// TwinCAT 3 PLC project Main
// ProgramVersion: 3.1.4023.0
// libraries:
//   mobject-fsm, * (mobject-io-ext)
//   Tc3_Module, * (Beckhoff Automation GmbH)
// project tree:
//   / PlcTask.TcTTO
//   Programs/ Main.TcPOU
//   TestMachine/ TestMachine.TcPOU, TestMachineEvents.TcDUT
// real-time tasks:
//   TASK PlcTask: cycle T#10ms, priority 20, ADS port 350

CONFIGURATION Main
    RESOURCE PLC ON TwinCAT3
        TASK PlcTask(INTERVAL := T#10ms, PRIORITY := 20);
        PROGRAM Main WITH PlcTask : Main;
    END_RESOURCE
END_CONFIGURATION

// ---- TestMachine/TestMachineEvents.TcDUT
{attribute 'qualified_only'}
{attribute 'strict'}
TYPE TestMachineEvents :
(
	Start,
	Stop,
	Abort,
	Reset,
	Clear
);
END_TYPE

// ---- Programs/Main.TcPOU
PROGRAM Main
VAR
	machine : TestMachine;
	currentState : STRING;
	start : BOOL;
	stop : BOOL;
	reset : BOOL;
	clear : BOOL;
	abort : BOOL;
END_VAR

IF start THEN
	start := FALSE;
	machine.Start();
END_IF

IF stop THEN
	stop := FALSE;
	machine.Stop();
END_IF

IF reset THEN
	reset := FALSE;
	machine.Reset();
END_IF

IF clear THEN
	clear := FALSE;
	machine.Clear();
END_IF

IF abort THEN
	abort := FALSE;
	machine.Abort();
END_IF

currentState := machine.CurrentStateName;

END_PROGRAM

// ---- TestMachine/TestMachine.TcPOU
FUNCTION_BLOCK TestMachine
VAR
	idleState : State(name := 'Idle');
	runningState : State(name := 'Running');
	stoppedState : State(name := 'Stopped');
	abortedState : State(name := 'Aborted');
	
	t2 : Transition(event := TestMachineEvents.Start, sourceState := idleState, destinationState := runningState);
	t1 : Transition(event := TestMachineEvents.Stop, sourceState := runningState, destinationState := stoppedState);
	t3 : Transition(event := TestMachineEvents.Abort, sourceState := idleState, destinationState := abortedState);
	t4 : Transition(event := TestMachineEvents.Abort, sourceState := runningState, destinationState := abortedState);
	t5 : Transition(event := TestMachineEvents.Abort, sourceState := stoppedState, destinationState := abortedState);
	t6 : Transition(event := TestMachineEvents.Reset, sourceState := stoppedState, destinationState := idleState);
	t7 : Transition(event := TestMachineEvents.Clear, sourceState := abortedState, destinationState := IdleState);
	
	tl1 : TransitionList(t1, 0);
	tl2 : TransitionList(t2, tl1);
	tl3 : TransitionList(t3, tl2);
	tl4 : TransitionList(t4, tl3);
	tl5 : TransitionList(t5, tl4);
	tl6 : TransitionList(t6, tl5);
	tl7 : TransitionList(t7, tl6);
	
	fsm : FSM(defaultState := idleState, transitions := tl7);
END_VAR

METHOD Abort
VAR_INPUT
END_VAR
fsm.Event(TestMachineEvents.Abort);
END_METHOD

METHOD Clear
fsm.Event(TestMachineEvents.Clear);
END_METHOD

PROPERTY CurrentStateName : STRING
GET
CurrentStateName := fsm.CurrentState.Name;
END_GET
END_PROPERTY

METHOD Reset
fsm.Event(TestMachineEvents.Reset);
END_METHOD

METHOD Start
fsm.Event(TestMachineEvents.Start);
END_METHOD

METHOD Stop
fsm.Event(TestMachineEvents.Stop);
END_METHOD

END_FUNCTION_BLOCK
